// TIA Portal project "2022.06.04_电机急停" (V17)

(* hardware
DEVICE "S7-1200 station_1"  S7-1200 Station
   slot 0: "Rack_0"  S7-1200 Rack  Rack  V1.0
   slot 1: "PLC_1"  CPU 1212C DC/DC/DC  6ES7 212-1AE40-0XB0  V4.5
*)

// ===== PLC "PLC_1"  CPU 1212C DC/DC/DC =====

VAR_GLOBAL   // PLC tag table "默认变量表"
   "启动" AT %I0.0 : Bool;
   "电机" AT %Q0.0 : Bool;
   "急停" AT %I0.1 : Bool;
   "重设时间" AT %I0.2 : Bool;
   "散热" AT %Q0.1 : Bool;
   "Tag_1" AT %I0.3 : Bool;
   "Tag_2" AT %Q0.2 : Bool;
   "Tag_3" AT %I0.4 : Bool;
   "Tag_4" AT %Q0.3 : Bool;
   "Tag_5" AT %MD0 : Time;
END_VAR

// folder: System blocks/Program resources

DATA_BLOCK "IEC_Timer_0_DB"   // DB1
{ S7_Optimized_Access := 'TRUE' }
AUTHOR : Simatic
FAMILY : IEC
NAME : IEC_TMR
VERSION : 1.0
// stored: InstanceOfName IEC_TIMER
"IEC_TIMER"
BEGIN
END_DATA_BLOCK

DATA_BLOCK "IEC_Timer_0_DB_1"   // DB2
{ S7_Optimized_Access := 'TRUE' }
AUTHOR : Simatic
FAMILY : IEC
NAME : IEC_TMR
VERSION : 1.0
// stored: InstanceOfName IEC_TIMER
"IEC_TIMER"
BEGIN
END_DATA_BLOCK

DATA_BLOCK "IEC_Timer_0_DB_2"   // DB3
{ S7_Optimized_Access := 'TRUE' }
AUTHOR : Simatic
FAMILY : IEC
NAME : IEC_TMR
VERSION : 1.0
// stored: InstanceOfName IEC_TIMER
"IEC_TIMER"
BEGIN
END_DATA_BLOCK

// folder: (top level)

ORGANIZATION_BLOCK "Main"   // OB1, LAD, ProgramCycle
TITLE = "Main Program Sweep (Cycle)"
{ S7_Optimized_Access := 'TRUE' }
VERSION : 0.1
   VAR_INPUT
      Initial_Call : Bool;   // Initial call of this OB
      Remanence : Bool;   // =True, if remanent data are available
   END_VAR
BEGIN

REGION Network 1
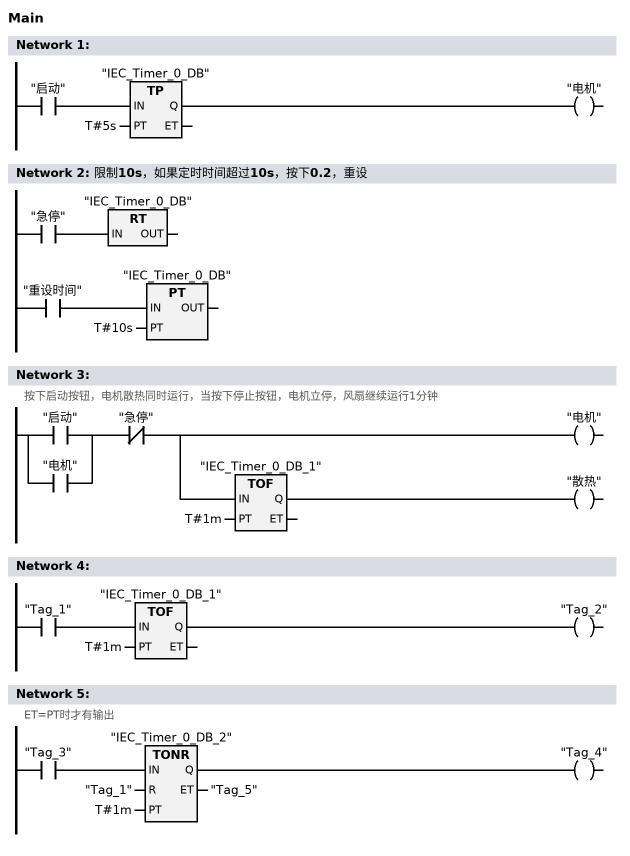
   "IEC_Timer_0_DB".TP(IN := "启动", PT := T#5s);
   "电机" := "IEC_Timer_0_DB".Q;
END_REGION

REGION Network 2: 限制10s，如果定时时间超过10s，按下0.2，重设
   IF "急停" THEN RESET_TIMER("IEC_Timer_0_DB"); END_IF;
   IF "重设时间" THEN PRESET_TIMER(PT := T#10s, TIMER := "IEC_Timer_0_DB"); END_IF;
END_REGION

REGION Network 3
   // 按下启动按钮，电机散热同时运行，当按下停止按钮，电机立停，风扇继续运行1分钟
   "电机" := ("启动" OR "电机") AND NOT "急停";
   "IEC_Timer_0_DB_1".TOF(IN := "电机", PT := T#1m);
   "散热" := "IEC_Timer_0_DB_1".Q;
END_REGION

REGION Network 4
   "IEC_Timer_0_DB_1".TOF(IN := "Tag_1", PT := T#1m);
   "Tag_2" := "IEC_Timer_0_DB_1".Q;
END_REGION

REGION Network 5
   // ET=PT时才有输出
   "IEC_Timer_0_DB_2".TONR(IN := "Tag_3", R := "Tag_1", PT := T#1m, ET => "Tag_5");
   "Tag_4" := "IEC_Timer_0_DB_2".Q;
END_REGION
END_ORGANIZATION_BLOCK